(* PLC project KinIn_v3.project, CODESYS CODESYS V3.5 SP19 *)
(* stored: creationDateTime 2025-01-20T16:24:05.1029997, modificationDateTime 2025-01-20T16:17:39.6822999 *)

FUNCTION_BLOCK expToRotAxisAndAngle
  VAR
    i : DINT;
    norm : norm;
    norm_expc3 : REAL;
  END_VAR
  VAR_INPUT
    {attribute 'variable_length_array_original_scope' := 'Inout'}
    {attribute 'variable_length_array' := 'ARRAY[*] OF REAL'}
    {attribute 'Dimensions' := '1'}
    expc3 : POINTER TO REAL;  (* vector *)
  END_VAR
  VAR_OUTPUT
    omghat : ARRAY[1..3] OF REAL;  (* scalar *)
    theta : REAL;
  END_VAR

            norm(vector:=expc3,
		normValue=>theta);
FOR i:= 1 TO UPPER_BOUND(expc3,1)DO
	omghat[i] :=expc3[i]/theta;
END_FOR

          
END_FUNCTION_BLOCK
